{attribute 'linkalways'} 
{attribute 'no_explicit_call' := 'This FB is a CLASS and must be accessed using methods or properties'}
{attribute 'enable_dynamic_creation'}
FUNCTION_BLOCK Node_F_VN_KeyPointsAndDescriptorsBRISK EXTENDS VisionNode
VAR
    ipSrcImage : _ITcVnImage;
    ipKeyPoints : _ITcVnContainer;
    ipDescriptors : _ITcVnImage;
    hrPrev : _HRESULT(S_OK);
	hresult : _HRESULT(S_OK);
END_VAR

METHOD PUBLIC  Clone : I_Node
VAR
	pNode : POINTER TO Node_F_VN_KeyPointsAndDescriptorsBRISK;
END_VAR
pNode := __NEW(Node_F_VN_KeyPointsAndDescriptorsBRISK);
Clone := pNode^;
END_METHOD

METHOD FB_init : BOOL
VAR_INPUT
	bInitRetains : BOOL; // if TRUE, the retain variables are initialized (warm start / cold start)
	bInCopyCode : BOOL;  // if TRUE, the instance afterwards gets moved into the copy code (online change)
END_VAR
AddInput('ipSrcImage', ipSrcImage);
AddInput('hrPrev', hrPrev);
AddOutput('ipKeyPoints', ipKeyPoints);
AddOutput('ipDescriptors', ipDescriptors);
AddOutput('hresult',hresult);
END_METHOD

METHOD PROTECTED OnExecute
hresult.Value := F_VN_KeyPointsAndDescriptorsBRISK(
	ipSrcImage := ipSrcImage.Value,
    ipKeyPoints := ipKeyPoints.Value,
    ipDescriptors := ipDescriptors.Value,
	hrPrev:= hrPrev.Value);
END_METHOD

METHOD PUBLIC PreExecutionCheck
VAR_INPUT
	Check : I_PreExecutionChecks;
END_VAR
Check.IsTrue(ipSrcImage.IsValid, 'ipSrcImage must contain an image');
Check.IsTrue(ipSrcImage.HasChannelCount(1), 'ipSrcImage must have 1 channel');
END_METHOD

END_FUNCTION_BLOCK

(* stored: Version 1.1.0.1, ProductVersion 3.1.4024.15
   POU Node_F_VN_KeyPointsAndDescriptorsBRISK: Id {10953c1b-594e-035c-0ee3-7d8005161e5d}, SpecialFunc None
   Folder Constructor: Id {b94897a9-d90a-0a21-0221-fc39793ef822}
   Method Clone: Id {f4ab82e6-b31a-01e4-2108-823d4d8bda57}
   Method FB_init: Id {d769bf28-bc0e-0798-18f3-7012bd24ec10}
   Method OnExecute: Id {ebad247d-a9a7-0087-27b1-cf171d8cdd0d}
   Method PreExecutionCheck: Id {5f29c3c4-7360-0320-22f3-61020fa9c3c3} *)
